(* PLC project Blank Project, Blank Blank 1.0 *)
(* stored: creationDateTime 2016-05-18T21:14:07, modificationDateTime 2024-12-26T09:55:48 *)

PROGRAM My_Program
  VAR
    iniciar AT %IX0.0 : BOOL := TRUE;
    parar AT %IX0.1 : BOOL := TRUE;
    lamp AT %QX0.0 : BOOL;
  END_VAR

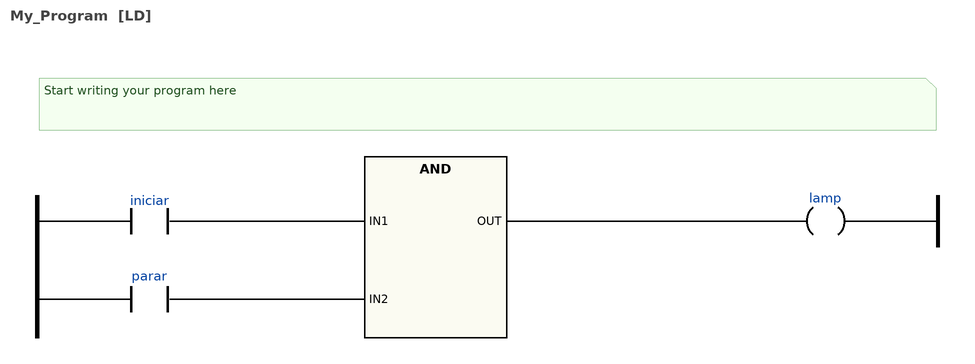
(* LD diagram, written out as Structured Text *)
(* Start writing your program here *)
lamp := iniciar AND parar;
END_PROGRAM

CONFIGURATION STD_CONF
  RESOURCE STD_RESSOURCE ON PLC
    TASK TaskMain(INTERVAL := T#50ms, PRIORITY := 0);
    PROGRAM Inst0 WITH TaskMain : My_Program;
  END_RESOURCE
END_CONFIGURATION
